PROGRAM Axe_02_ZChariot (*Chariot*)
VAR	RE_Cellule: R_TRIG;	ZChariot: FB_Axe_Ethercat_V2;		B_Fc_Origine_X_Chariot: BOOL;
		Defaut_Var_Chariot_AX5000: BOOL;
		Diag_Nbrs_Var_Chariot_AX5000 :UDINT;
		Diag_Mess_Var_Chariot_AX5000: STRING;


END_VAR

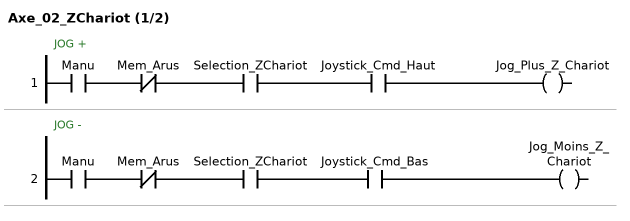
// NETWORK 1
// JOG +
Jog_Plus_Z_Chariot := Manu AND NOT Mem_Arus AND Selection_ZChariot AND Joystick_Cmd_Haut;

// NETWORK 2
// JOG -
Jog_Moins_Z_Chariot := Manu AND NOT Mem_Arus AND Selection_ZChariot AND Joystick_Cmd_Bas;

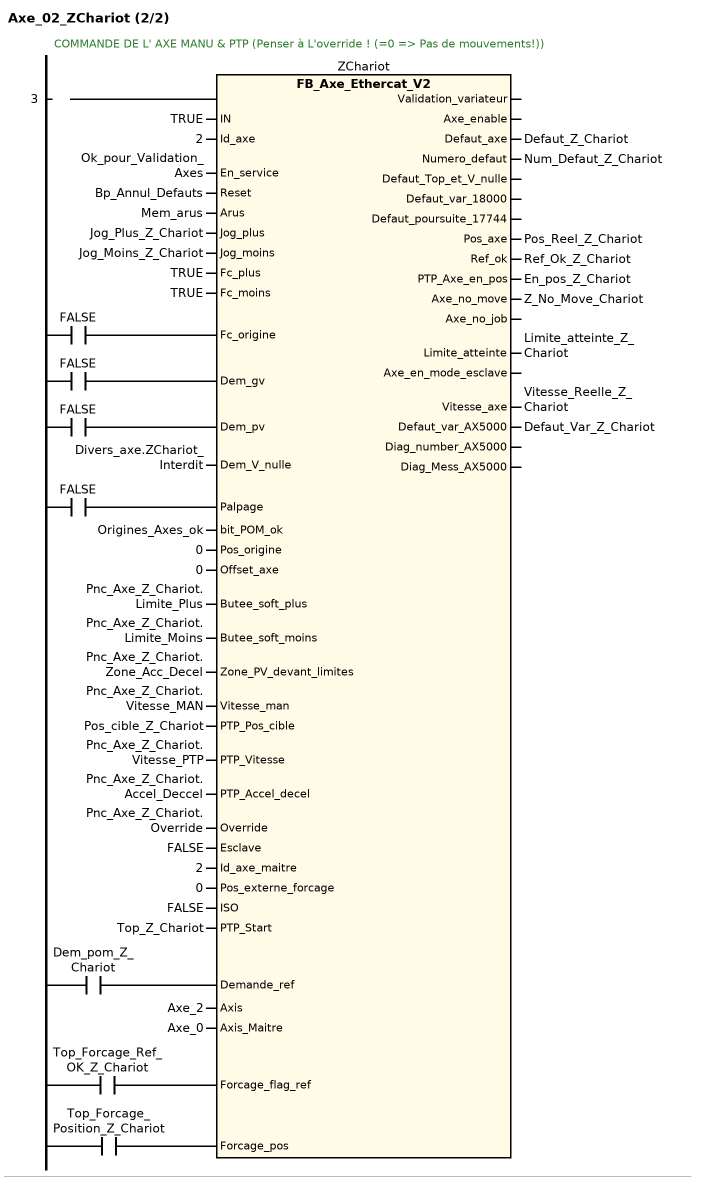
// NETWORK 3
// 					COMMANDE DE L' AXE MANU & PTP (Penser à L'override ! (=0 => Pas de mouvements!))
//
//
ZChariot(
    IN := TRUE,
    Id_axe := 2,
    En_service := Ok_pour_Validation_Axes,
    Reset := Bp_Annul_Defauts,
    Arus := Mem_arus,
    Jog_plus := Jog_Plus_Z_Chariot,
    Jog_moins := Jog_Moins_Z_Chariot,
    Fc_plus := TRUE,
    Fc_moins := TRUE,
    Fc_origine := FALSE,
    Dem_gv := FALSE,
    Dem_pv := FALSE,
    Dem_V_nulle := Divers_axe.ZChariot_Interdit,
    Palpage := FALSE,
    bit_POM_ok := Origines_Axes_ok,
    Pos_origine := 0,
    Offset_axe := 0,
    Butee_soft_plus := Pnc_Axe_Z_Chariot.Limite_Plus,
    Butee_soft_moins := Pnc_Axe_Z_Chariot.Limite_Moins,
    Zone_PV_devant_limites := Pnc_Axe_Z_Chariot.Zone_Acc_Decel,
    Vitesse_man := Pnc_Axe_Z_Chariot.Vitesse_MAN,
    PTP_Pos_cible := Pos_cible_Z_Chariot,
    PTP_Vitesse := Pnc_Axe_Z_Chariot.Vitesse_PTP,
    PTP_Accel_decel := Pnc_Axe_Z_Chariot.Accel_Deccel,
    Override := Pnc_Axe_Z_Chariot.Override,
    Esclave := FALSE,
    Id_axe_maitre := 2,
    Pos_externe_forcage := 0,
    ISO := FALSE,
    PTP_Start := Top_Z_Chariot,
    Demande_ref := Dem_pom_Z_Chariot,
    Axis := Axe_2,
    Axis_Maitre := Axe_0,
    Forcage_flag_ref := Top_Forcage_Ref_OK_Z_Chariot,
    Forcage_pos := Top_Forcage_Position_Z_Chariot,
    Defaut_axe => Defaut_Z_Chariot,
    Numero_defaut => Num_Defaut_Z_Chariot,
    Pos_axe => Pos_Reel_Z_Chariot,
    Ref_ok => Ref_Ok_Z_Chariot,
    PTP_Axe_en_pos => En_pos_Z_Chariot,
    Axe_no_move => Z_No_Move_Chariot,
    Limite_atteinte => Limite_atteinte_Z_Chariot,
    Vitesse_axe => Vitesse_Reelle_Z_Chariot,
    Defaut_var_AX5000 => Defaut_Var_Z_Chariot); // FB_Axe_Ethercat_V2

END_PROGRAM

(* stored: Version 1.1.0.1, ProductVersion 3.1.4024.15
   POU Axe_02_ZChariot: Id {86a6316a-8779-449b-a257-59b3a721b002}, SpecialFunc None *)
